// TIA Portal V17 export
// export: Created 2023-02-14T02:49:47.8292955Z, ExportSetting WithDefaults, DisplayName Totally Integrated Automation Portal, DisplayVersion V17, DisplayName TIA Portal Openness, DisplayVersion V17, DisplayName TIA Portal Teamcenter Gateway, DisplayVersion V17, DisplayName TIA Portal Version Control Interface, DisplayVersion V17, DisplayName SINAMICS Startdrive Advanced, DisplayVersion V17, DisplayName SINAMICS Startdrive G130, G150, S120, S150, SINAMICS MV, S210, DisplayVersion V17, DisplayName SINAMICS Startdrive G110M, G120, G120C, G120D, G120P, G115D, DisplayVersion V17, DisplayName STEP 7 Professional, DisplayVersion V17, DisplayName STEP 7 Safety, DisplayVersion V17, DisplayName WinCC Professional, DisplayVersion V17
DATA_BLOCK "BFT-66"   // DB114
VERSION : 0.1
// stored: AutoNumber false, DBAccessibleFromOPCUA true, DBAccessibleFromWebserver true, InstanceOfName Buffer_Tank, InstanceOfType FB
"Buffer_Tank"
   // VAR_INPUT
   //    IN_LT01 : Real;
   //    "Tank w Circulation" : Bool;
   //    AlarmProd_pasteur : Bool;
   //    HighLevel_pasteur : Bool;
   //    IN_FBAV_Inload : Bool;
   //    IN_FBAV_CIP_Tank : Bool;
   //    IN_FBAV_CIP_Line : Bool;
   //    IN_FBAV_Outlet : Bool;
   //    IN_FBAV_Transfer : Bool;
   //    IN_FBP_Transfer : Bool;
   //    IN_FBXA : Bool;
   //    IN_FBP_Circulation : Bool;
   //    IN_Product_Ready : Bool;
   //    IN_Product_TransferOnProg : Bool;
   //    "Inload Busy" : Bool;
   //    "CIP Pulse" : Bool;
   //    "CIP Req OK" : Bool;
   //    "CIP Supply ON" : Bool;
   //    "CIP In Progress" : Bool;
   //    "CIP Complete" : Bool;
   //    "CIP Busy" : Bool;
   // END_VAR
   // VAR_OUTPUT
   //    Out_AV_Inload : Bool;
   //    Out_AV_Drain_In : Bool;
   //    Out_AV_CIP_Tank : Bool;
   //    Out_AV_CIP_Line : Bool;
   //    Out_AV_Outlet : Bool;
   //    Out_AV_Transfer : Bool;
   //    Out_P_Transfer : Bool;
   //    Out_P_Transfer_SP : Real;
   //    Out_XA : Bool;
   //    Out_XA_SP : Real;
   //    Out_P_Circulation : Bool;
   //    Out_Prod_Req : Bool;
   //    Out_Prod_LineOpen : Bool;
   //    Out_CIP_Tank_Req : Bool;
   //    Out_CIP_Line_Req : Bool;
   //    Out_CIP_Tank_LineOpen : Bool;
   //    Out_CIP_Line_LineOpen : Bool;
   // END_VAR
   // VAR
   //    cmd : Struct
   //       Inload : Bool;
   //       Drain_In : Bool;
   //       Ready_for_Transfer : Bool;
   //       CIP_Tank : Bool;
   //       CIP_Line : Bool;
   //       Agitator_Mode : Bool;
   //       Agitator_Man_OnOff : Bool;
   //       Agitator_SpeedMode : Bool;
   //       Circulation : Bool;
   //    END_STRUCT;
   // END_VAR
   // VAR RETAIN
   //    param : Struct
   //       L_Lo_Lim : Real;
   //       L_Hi_Lim : Real;
   //       L_Hys : Real;
   //       "Circulation Level" : Real;
   //       SP_Level_HL : Real;
   //       SP_Level_ML : Real;
   //       SP_Level_LL : Real;
   //       DrainIn : DInt;
   //       SP_Pump_Transfer : Real;
   //       SP_Pump_CIP : Real;
   //       SP_Agitator : Real;
   //       SP_Level_Agi_ON1 : Real;
   //       SP_Level_Agi_OFF1 : Real;
   //       SP_Level_Agi_ON2 : Real;
   //       SP_Level_Agi_OFF2 : Real;
   //       SP_Level_Agi_ON3 : Real;
   //       "CIP Ret On" : Real;
   //       "CIP Ret Off" : Real;
   //    END_STRUCT;
   // END_VAR
   // VAR
   //    state : Struct
   //       "Tank LL" : Bool;
   //       "Tank ML" : Bool;
   //       "Tank HL" : Bool;
   //       "Tank CIP En" : Bool;
   //       "Tank CIP" : Bool;
   //       "Line CIP En" : Bool;
   //       "Line CIP" : Bool;
   //       "Ready for Transfer En" : Bool;
   //       "Ready for Transfer" : Bool;
   //       Inloading : Bool;
   //       "Inload En" : Bool;
   //       L_Agi_ON1 : Bool;
   //       L_Agi_ON2 : Bool;
   //       L_Agi_ON3 : Bool;
   //       Tank_Circulation : Bool;
   //       "Circulation Enable" : Bool;
   //       Circulation : Bool;
   //       "Transfer on Prog" : Bool;
   //       "CIP Return On" : Bool;
   //       "CIP Req" : Bool;
   //    END_STRUCT;
   //    alwaysOn : Bool;
   //    L_Hys_Abs : Real;
   //    Hys_Level_LL : Real;
   //    Hys_Level_ML : Real;
   //    Hys_Level_HL : Real;
   //    Hys_Level_Circ : Real;
   //    r : Struct
   //       PosE1 : Bool;
   //       PosE2 : Bool;
   //       PosE3 : Bool;
   //       PosE4 : Bool;
   //       PosE5 : Bool;
   //       PosE6 : Bool;
   //       PosE7 : Bool;
   //       PosE8 : Bool;
   //       PosE9 : Bool;
   //       PosE10 : Bool;
   //       PosE11 : Bool;
   //       PosE12 : Bool;
   //       PosE13 : Bool;
   //       PosE14 : Bool;
   //       PosE15 : Bool;
   //       PosE16 : Bool;
   //       PosE17 : Bool;
   //       PosE18 : Bool;
   //       PosE19 : Bool;
   //       PosE20 : Bool;
   //       PosE21 : Bool;
   //       PosE22 : Bool;
   //       PosE23 : Bool;
   //       PosE24 : Bool;
   //       PosE25 : Bool;
   //       PosE26 : Bool;
   //       PosE27 : Bool;
   //       PosE28 : Bool;
   //       PosE29 : Bool;
   //       PosE30 : Bool;
   //       PosE31 : Bool;
   //       PosE32 : Bool;
   //    END_STRUCT;
   //    Actuator : Struct
   //       AV_Inload : Bool;
   //       AV_Drain_In : Bool;
   //       AV_Outlet : Bool;
   //       AV_Transfer : Bool;
   //       AV_CIP_Tank : Bool;
   //       AV_CIP_Line : Bool;
   //       P_Transfer : Bool;
   //       P_CIP : Bool;
   //       Agitator_level : Bool;
   //    END_STRUCT;
   //    DrainIn_OnTime : TON_TIME;
   //    DrainIn_OffTime : TOF_TIME;
   //    InloadAV_OffTime : TOF_TIME;
   //    DrainIn_MS : DInt;
   //    L_AgiTim : TON_TIME;
   // END_VAR
BEGIN
END_DATA_BLOCK
